{attribute 'no_explicit_call' := 'do not call this function block directly'} 
{attribute 'enable_dynamic_creation'}
FUNCTION_BLOCK PointerUniqueSetEnumerator EXTENDS Enumerator
VAR
	_ClassName : STRING := __POUNAME();
	_HashSet : IReadOnlyPointerUniqueSet;
	_Current : PVOID;
END_VAR

{attribute 'monitoring' := 'call'}
PROPERTY ClassName : STRING
GET
ClassName := _ClassName;
END_GET
END_PROPERTY

{attribute 'OPC.UA.DA.Property' := '1'}
{attribute 'monitoring' := 'call'}
PROPERTY Current : PVOID
GET
Current := ADR(_Current);
END_GET
END_PROPERTY

METHOD INTERNAL Initialize 
VAR_INPUT
	hashSet : IReadOnlyPointerUniqueSet;
END_VAR
_HashSet := hashSet;
END_METHOD

{attribute "object_name" := "MoveNext"}
METHOD MoveNext : BOOL
_CurrentIndex := _CurrentIndex + 1;

IF _CurrentIndex >= _HashSet.Count THEN
	_Current := 0;
	_CurrentIndex := _HashSet.Count;
ELSE
	_Current := _HashSet.GetByIndex(_CurrentIndex);	
	MoveNext := TRUE;
END_IF
END_METHOD

{attribute "object_name" := "Reset"}
METHOD Reset
SUPER^.Reset();

_Current := 0;
END_METHOD

END_FUNCTION_BLOCK

(* stored: Version 1.1.0.1
   POU PointerUniqueSetEnumerator: Id {7acbb17a-360f-0678-260c-74eab69831f9}, SpecialFunc None
   Property ClassName: Id {707e3de4-04f8-0e50-0059-95c83de50d68}
   Get Get: Id {612a2437-bdd8-0bfa-14ca-37d056ba2705}
   Property Current: Id {efa29b5c-71b4-05b0-3b4b-a125f677b8b0}
   Get Get: Id {472543a4-15ef-0243-0b2f-68e80680922c}
   Method Initialize: Id {43c696b5-034c-0633-0eec-2d0a98be1e12}
   Method MoveNext: Id {f92f59b2-340b-0061-0837-15cf129df717}
   Method Reset: Id {a69a2270-26fd-0bda-2aed-31f55cf36e58} *)
